{attribute 'GeneratedUsingTerminal: EJ5002-0000-0016'}
{attribute addProperty BoxType "EJ5002-0000-0016"}
{attribute addProperty Id "EtcSlaveTerminalBaseSSI_Inputs_Channel_1AT %I*SSI_Inputs_Channel_0E3D8E3310SSI_Inputs_Channel_2AT %I*SSI_Inputs_Channel_0E3D8E3310WcStateAT %I*WcState_9091E0EB2InfoDataAT %I*InfoData_32EB74EA10"}
{attribute addProperty CRC "2169208955"}
{attribute addProperty Size "32"}
TYPE EJ5002_814B807B EXTENDS EtcSlaveTerminalBase :
STRUCT
	{attribute addProperty Name "SSI_Inputs_Channel_1"}
	SSI_Inputs_Channel_1 : SSI_Inputs_Channel_0E3D8E33;
	{attribute addProperty Name "SSI_Inputs_Channel_2"}
	SSI_Inputs_Channel_2 : SSI_Inputs_Channel_0E3D8E33;
	{attribute addProperty Name "WcState"}
	WcState : WcState_9091E0EB;
	{attribute addProperty Name "InfoData"}
	InfoData : InfoData_32EB74EA;
END_STRUCT
END_TYPE

(* stored: Version 1.2.0.0, ProductVersion 3.1.4024.9
   DUT EJ5002_814B807B: Id {94692b57-76eb-44b4-88d8-2924a778b517} *)
